{attribute 'qualified_only'}
VAR_GLOBAL CONSTANT
	NumberOfChildren : INT := 5;
END_VAR

(* stored: Version 1.1.0.1, ProductVersion 3.1.4024.12
   GVL Param: Id {d78f346c-9d30-4d6c-be7e-0bf931407fc1}, ParameterList True *)
